// global function to extract state identifier from combined value
FUNCTION f_GetState : uint
VAR_INPUT
  state     : UINT; // combined value of identifier + e_progress
END_VAR
VAR
  _stx      : uint;
END_VAR

_stx          := state MOD E_PROGRESS.PROGRESS_INIT;

IF (_stx = 0)
THEN
  f_GetState  := state;
ELSE
  f_GetState  := _stx;
END_IF

END_FUNCTION

(* stored: Version 1.1.0.1
   POU f_GetState: Id {4d4902ba-e5f9-48ad-9d1b-c8cb49982b26}, SpecialFunc None *)
